(* IEC 61131-3 sources: ArfBotOS/Codesys-4/ArfBotOS.fbsdev/Application.iecapp^/FUN/template/FB_Module.fb.st^/PropErrDescription.prop.st^, 1 file *)

(* ---- Get.meth.st ---- *)
VAR
END_VAR

PropErrDescription := ErrorDescription;
